(* IEC 61131-3 sources: POMIRTS_lab3/AS/Library_2/AsNxDpS, 3 files *)

(* ---- AsNxDpS.typ ---- *)
TYPE
	nxdpsAddAdrParam_t		: STRUCT			(*additional address parameter*)
		srcType				: USINT;
		srcSize				: USINT;
		destType			: USINT;
		destSize			: USINT;
		addParam			: ARRAY[0..227] OF USINT;
	END_STRUCT;

	nxdpsIm0_t				: STRUCT			(*I&M0 parameter*)
		manufactor			: ARRAY[0..9] OF USINT;
		manufactorId		: UINT;
		orderId				: ARRAY[0..19] OF USINT;
		serialNumber		: ARRAY[0..15] OF USINT;
		hwRevision			: UINT;
		swRevision			: ARRAY[0..3] OF USINT;
		revisionCounter		: UINT;
		profileId			: UINT;
		profileSpecType		: UINT;
		imVersion			: UINT;
		imSupported			: UINT;
	END_STRUCT;
END_TYPE

(* ---- AsNxDpS.fun ---- *)
{REDUND_CONTEXT} {REDUND_UNREPLICABLE} FUNCTION_BLOCK nxdpsSubscribe			(*subscribe slave*)
	VAR_INPUT
		enable			: BOOL;			(*enables execution*)
		pDevice			: UDINT;		(*interface name given as a pointer, e.g., "SL<x>.SS<y>.IF<z>"*)
	END_VAR
	VAR
        _state			: UINT;			(*internal variable*)
		_result			: UINT;			(*internal variable*)
        _srcId			: UDINT;		(*internal variable*)
	END_VAR
	VAR_OUTPUT
		status			: UINT;			(*execution status: ERR_OK, ERR_FUB_ENABLE_FALSE, ERR_FUB_BUSY, 0xXXXX = see help*)
		dpStatus		: UDINT;		(*profibus DP stack status*)
	END_VAR
END_FUNCTION_BLOCK

{REDUND_CONTEXT} {REDUND_UNREPLICABLE} FUNCTION_BLOCK nxdpsUnsubscribe			(*unsubscribe slave*)
	VAR_INPUT
		enable			: BOOL;			(*enables execution*)
		pDevice			: UDINT;		(*interface name given as a pointer, e.g., "SL<x>.SS<y>.IF<z>"*)
	END_VAR
	VAR
        _state			: UINT;			(*internal variable*)
		_result			: UINT;			(*internal variable*)
        _srcId			: UDINT;		(*internal variable*)
	END_VAR
	VAR_OUTPUT
		status			: UINT;			(*execution status: ERR_OK, ERR_FUB_ENABLE_FALSE, ERR_FUB_BUSY, 0xXXXX = see help*)
		dpStatus		: UDINT;		(*profibus DP stack status*)
	END_VAR
END_FUNCTION_BLOCK

{REDUND_CONTEXT} {REDUND_UNREPLICABLE} FUNCTION_BLOCK nxdpsAlarmNotification	(*alarm notification*)
	VAR_INPUT
		enable			: BOOL;			(*enables execution*)
		pDevice			: UDINT;		(*interface name given as a pointer, e.g., "SL<x>.SS<y>.IF<z>"*)
		slotNumber		: USINT;		(*slot number*)
		seqNumber		: USINT;		(*sequence number*)
		alarmType		: USINT;		(*alarm type*)
		alarmSpecifier	: USINT;		(*alarm specifier*)
		addAck			: BOOL;			(*additional acknowledgement flag*)
		alarmDataLen	: USINT;		(*alarm data length*)
		pAlarmData		: UDINT;		(*alarm data given as a pointer*)
	END_VAR
	VAR
        _state			: UINT;			(*internal variable*)
		_result			: UINT;			(*internal variable*)
        _srcId			: UDINT;		(*internal variable*)
	END_VAR
	VAR_OUTPUT
		status			: UINT;			(*execution status: ERR_OK, ERR_FUB_ENABLE_FALSE, ERR_FUB_BUSY, 0xXXXX = see help*)
		dpStatus		: UDINT;		(*profibus DP stack status*)
	END_VAR
END_FUNCTION_BLOCK

{REDUND_CONTEXT} {REDUND_UNREPLICABLE} FUNCTION_BLOCK nxdpsAlarmAckReceive		(*receive alarm acknowledgement*)
	VAR_INPUT
		enable			: BOOL;			(*enables execution*)
		pDevice			: UDINT;		(*interface name given as a pointer, e.g., "SL<x>.SS<y>.IF<z>"*)
	END_VAR
	VAR
        _state			: UINT;			(*internal variable*)
		_result			: UINT;			(*internal variable*)
        _srcId			: UDINT;		(*internal variable*)
	END_VAR
	VAR_OUTPUT
		status			: UINT;			(*execution status: ERR_OK, ERR_FUB_ENABLE_FALSE, ERR_FUB_BUSY, 0xXXXX = see help*)
		dpStatus		: UDINT;		(*profibus DP stack status*)
		slotNumber		: USINT;		(*slot number*)
		seqNumber		: USINT;		(*sequence number*)
		alarmType		: USINT;		(*alarm type*)
	END_VAR
END_FUNCTION_BLOCK

{REDUND_CONTEXT} {REDUND_UNREPLICABLE} FUNCTION_BLOCK nxdpsV1C1WriteInd		(*V1 class 1 write indication*)
	VAR_INPUT
		enable			: BOOL;			(*enables execution*)
		pDevice			: UDINT;		(*interface name given as a pointer, e.g., "SL<x>.SS<y>.IF<z>"*)
		maxDataLen		: UDINT;		(*max data length*)
		pData			: UDINT;		(*data buffer given as a pointer*)
	END_VAR
	VAR
        _state			: UINT;			(*internal variable*)
		_result			: UINT;			(*internal variable*)
        _srcId			: UDINT;		(*internal variable*)
	END_VAR
	VAR_OUTPUT
		status			: UINT;			(*execution status: ERR_OK, ERR_FUB_ENABLE_FALSE, ERR_FUB_BUSY, 0xXXXX = see help*)
		dpStatus		: UDINT;		(*profibus DP stack status*)
		slotNumber		: USINT;		(*slot number*)
		index			: USINT;		(*index*)
		dataLen			: USINT;		(*data length*)
		source			: UDINT;		(*source*)
		sourceId		: UDINT;		(*source id*)
	END_VAR
END_FUNCTION_BLOCK

{REDUND_CONTEXT} {REDUND_UNREPLICABLE} FUNCTION_BLOCK nxdpsV1C1WriteAck		(*V1 class 1 write acknowledgement*)
	VAR_INPUT
		enable			: BOOL;			(*enables execution*)
		pDevice			: UDINT;		(*interface name given as a pointer, e.g., "SL<x>.SS<y>.IF<z>"*)
		ackType			: BOOL;			(*type of acknowledgement*)
		slotNumber		: USINT;		(*slot number*)
		index			: USINT;		(*index*)
		dataLen			: USINT;		(*data length*)
		errorDecode		: USINT;		(*error decode*)
		errorCode1		: USINT;		(*error code 1*)
		errorCode2		: USINT;		(*error code 2*)
		source			: UDINT;		(*source*)
		sourceId		: UDINT;		(*source id*)
	END_VAR
	VAR
        _state			: UINT;			(*internal variable*)
		_result			: UINT;			(*internal variable*)
        _srcId			: UDINT;		(*internal variable*)
	END_VAR
	VAR_OUTPUT
		status			: UINT;			(*execution status: ERR_OK, ERR_FUB_ENABLE_FALSE, ERR_FUB_BUSY, 0xXXXX = see help*)
		dpStatus		: UDINT;		(*profibus DP stack status*)
	END_VAR
END_FUNCTION_BLOCK

{REDUND_CONTEXT} {REDUND_UNREPLICABLE} FUNCTION_BLOCK nxdpsV1C1ReadInd			(*V1 class 1 read indication*)
	VAR_INPUT
		enable			: BOOL;			(*enables execution*)
		pDevice			: UDINT;		(*interface name given as a pointer, e.g., "SL<x>.SS<y>.IF<z>"*)
	END_VAR
	VAR
        _state			: UINT;			(*internal variable*)
		_result			: UINT;			(*internal variable*)
        _srcId			: UDINT;		(*internal variable*)
	END_VAR
	VAR_OUTPUT
		status			: UINT;			(*execution status: ERR_OK, ERR_FUB_ENABLE_FALSE, ERR_FUB_BUSY, 0xXXXX = see help*)
		dpStatus		: UDINT;		(*profibus DP stack status*)
		slotNumber		: USINT;		(*slot number*)
		index			: USINT;		(*index*)
		dataLen			: USINT;		(*data length*)
		source			: UDINT;		(*source*)
		sourceId		: UDINT;		(*source id*)
	END_VAR
END_FUNCTION_BLOCK

{REDUND_CONTEXT} {REDUND_UNREPLICABLE} FUNCTION_BLOCK nxdpsV1C1ReadAck			(*V1 class 1 read acknowledgement*)
	VAR_INPUT
		enable			: BOOL;			(*enables execution*)
		pDevice			: UDINT;		(*interface name given as a pointer, e.g., "SL<x>.SS<y>.IF<z>"*)
		ackType			: BOOL;			(*type of acknowledgement*)
		slotNumber		: USINT;		(*slot number*)
		index			: USINT;		(*index*)
		dataLen			: USINT;		(*data length*)
		errorDecode		: USINT;		(*error decode*)
		errorCode1		: USINT;		(*error code 1*)
		errorCode2		: USINT;		(*error code 2*)
		source			: UDINT;		(*source*)
		sourceId		: UDINT;		(*source id*)
		pData			: UDINT;		(*data buffer given as pointer*)
	END_VAR
	VAR
        _state			: UINT;			(*internal variable*)
		_result			: UINT;			(*internal variable*)
        _srcId			: UDINT;		(*internal variable*)
	END_VAR
	VAR_OUTPUT
		status			: UINT;			(*execution status: ERR_OK, ERR_FUB_ENABLE_FALSE, ERR_FUB_BUSY, 0xXXXX = see help*)
		dpStatus		: UDINT;		(*profibus DP stack status*)
	END_VAR
END_FUNCTION_BLOCK

{REDUND_CONTEXT} {REDUND_UNREPLICABLE} FUNCTION_BLOCK nxdpsSetDiag				(*set diagnostic*)
	VAR_INPUT
		enable			: BOOL;			(*enables execution*)
		pDevice			: UDINT;		(*interface name given as a pointer, e.g., "SL<x>.SS<y>.IF<z>"*)
		extDiag			: BOOL;			(*extended diagnostic*)
		extDiagOverflow	: BOOL;			(*extended diagnostic overflow*)
		pDiagData		: UDINT;		(*diagnostic data given as a pointer*)
		diagDataLen		: UDINT;		(*diagnostic data length*)
	END_VAR
	VAR
        _state			: UINT;			(*internal variable*)
		_result			: UINT;			(*internal variable*)
        _srcId			: UDINT;		(*internal variable*)
	END_VAR
	VAR_OUTPUT
		status			: UINT;			(*execution status: ERR_OK, ERR_FUB_ENABLE_FALSE, ERR_FUB_BUSY, 0xXXXX = see help*)
		dpStatus		: UDINT;		(*profibus DP stack status*)
	END_VAR
END_FUNCTION_BLOCK

{REDUND_CONTEXT} {REDUND_UNREPLICABLE} FUNCTION_BLOCK nxdpsSetIm0				(*change I&M0 parameter settings*)
	VAR_INPUT
		enable				: BOOL;			(*enables execution*)
		pDevice				: UDINT;		(*interface name given as a pointer, e.g., "SL<x>.SS<y>.IF<z>"*)
		im0Param			: nxdpsIm0_t;	(*I&M0 parameter*)
		profSpecSupp		: BOOL;
		manuSpecSupp		: BOOL;
		slotsNotZeroSupp	: BOOL;
	END_VAR
	VAR
        _state			: UINT;			(*internal variable*)
		_result			: UINT;			(*internal variable*)
        _srcId			: UDINT;		(*internal variable*)
	END_VAR
	VAR_OUTPUT
		status			: UINT;			(*execution status: ERR_OK, ERR_FUB_ENABLE_FALSE, ERR_FUB_BUSY, 0xXXXX = see help*)
		dpStatus		: UDINT;		(*profibus DP stack status*)
	END_VAR
END_FUNCTION_BLOCK

{REDUND_CONTEXT} {REDUND_UNREPLICABLE} FUNCTION_BLOCK nxdpsSetAdr				(*set address*)
	VAR_INPUT
		enable			: BOOL;			(*enables execution*)
		pDevice			: UDINT;		(*interface name given as a pointer, e.g., "SL<x>.SS<y>.IF<z>"*)
		address			: UDINT;		(*new slave address*)
	END_VAR
	VAR
        _state			: UINT;			(*internal variable*)
		_result			: UINT;			(*internal variable*)
        _srcId			: UDINT;		(*internal variable*)
	END_VAR
	VAR_OUTPUT
		status			: UINT;			(*execution status: ERR_OK, ERR_FUB_ENABLE_FALSE, ERR_FUB_BUSY, 0xXXXX = see help*)
		dpStatus		: UDINT;		(*profibus DP stack status*)
	END_VAR
END_FUNCTION_BLOCK

{REDUND_CONTEXT} {REDUND_UNREPLICABLE} FUNCTION_BLOCK nxdpsStartBusComm		(*start bus communication*)
	VAR_INPUT
		enable			: BOOL;			(*enables execution*)
		pDevice			: UDINT;		(*interface name given as a pointer, e.g., "SL<x>.SS<y>.IF<z>"*)
	END_VAR
	VAR
        _state			: UINT;			(*internal variable*)
		_result			: UINT;			(*internal variable*)
        _srcId			: UDINT;		(*internal variable*)
	END_VAR
	VAR_OUTPUT
		status			: UINT;			(*execution status: ERR_OK, ERR_FUB_ENABLE_FALSE, ERR_FUB_BUSY, 0xXXXX = see help*)
		dpStatus		: UDINT;		(*profibus DP stack status*)
	END_VAR
END_FUNCTION_BLOCK

{REDUND_CONTEXT} {REDUND_UNREPLICABLE} FUNCTION_BLOCK nxdpsV1C2InitiateInd		(*V1 class2 initiate connection indication*)
	VAR_INPUT
		enable			: BOOL;			(*enables execution*)
		pDevice			: UDINT;		(*interface name given as a pointer, e.g., "SL<x>.SS<y>.IF<z>"*)
		pAddAdrParam	: UDINT;		(*additional address parameter table given as pointer*)
	END_VAR
	VAR
        _state			: UINT;			(*internal variable*)
		_result			: UINT;			(*internal variable*)
        _srcId			: UDINT;		(*internal variable*)
	END_VAR
	VAR_OUTPUT
		status			: UINT;			(*execution status: ERR_OK, ERR_FUB_ENABLE_FALSE, ERR_FUB_BUSY, 0xXXXX = see help*)
		dpStatus		: UDINT;		(*profibus DP stack status*)
		connectionRef	: UDINT;		(*connection reference*)
		featuresSup		: UINT;			(*requested featrures of the DP master class 2 connection*)
		profileFeatSup	: UINT;			(*requested profile featrures of the DP master class 2 connection*)
		profileIdent	: UINT;			(*profile ident number*)
		source			: UDINT;		(*source*)
		sourceId		: UDINT;		(*source id*)
	END_VAR
END_FUNCTION_BLOCK

{REDUND_CONTEXT} {REDUND_UNREPLICABLE} FUNCTION_BLOCK nxdpsV1C2InitiateRes		(*V1 class 2 initiate connection response*)
	VAR_INPUT
		enable			: BOOL;			(*enables execution*)
		pDevice			: UDINT;		(*interface name given as a pointer, e.g., "SL<x>.SS<y>.IF<z>"*)
		ackType			: BOOL;			(*type of acknowledgement*)
		connectionRef	: UDINT;		(*connection reference*)
		dataUnitSizeMax	: USINT;		(*maximum size of data unit to transfer*)
		featuresSup		: UINT;			(*requested featrures of the DP master class 2 connection*)
		profileFeatSup	: UINT;			(*requested profile featrures of the DP master class 2 connection*)
		profileIdent	: UINT;			(*profile ident number*)
		pAddAdrParam	: UDINT;		(*additional address parameter table given as pointer*)
		errorDecode		: USINT;		(*error decode*)
		errorCode1		: USINT;		(*error code 1*)
		errorCode2		: USINT;		(*error code 2*)
		source			: UDINT;		(*source*)
		sourceId		: UDINT;		(*source id*)
	END_VAR
	VAR
        _state			: UINT;			(*internal variable*)
		_result			: UINT;			(*internal variable*)
        _srcId			: UDINT;		(*internal variable*)
	END_VAR
	VAR_OUTPUT
		status			: UINT;			(*execution status: ERR_OK, ERR_FUB_ENABLE_FALSE, ERR_FUB_BUSY, 0xXXXX = see help*)
		dpStatus		: UDINT;		(*profibus DP stack status*)
	END_VAR
END_FUNCTION_BLOCK

{REDUND_CONTEXT} {REDUND_UNREPLICABLE} FUNCTION_BLOCK nxdpsV1C2ReadInd			(*V1 class 2 read indication*)
	VAR_INPUT
		enable			: BOOL;			(*enables execution*)
		pDevice			: UDINT;		(*interface name given as a pointer, e.g., "SL<x>.SS<y>.IF<z>"*)
	END_VAR
	VAR
        _state			: UINT;			(*internal variable*)
		_result			: UINT;			(*internal variable*)
        _srcId			: UDINT;		(*internal variable*)
	END_VAR
	VAR_OUTPUT
		status			: UINT;			(*execution status: ERR_OK, ERR_FUB_ENABLE_FALSE, ERR_FUB_BUSY, 0xXXXX = see help*)
		dpStatus		: UDINT;		(*profibus DP stack status*)
		connectionRef	: UDINT;		(*connection reference*)
		slotNumber		: USINT;		(*slot number*)
		index			: USINT;		(*index*)
		dataLen			: USINT;		(*data length*)
		source			: UDINT;		(*source*)
		sourceId		: UDINT;		(*source id*)
	END_VAR
END_FUNCTION_BLOCK

{REDUND_CONTEXT} {REDUND_UNREPLICABLE} FUNCTION_BLOCK nxdpsV1C2ReadRes			(*V1 class 2 read response*)
	VAR_INPUT
		enable			: BOOL;			(*enables execution*)
		pDevice			: UDINT;		(*interface name given as a pointer, e.g., "SL<x>.SS<y>.IF<z>"*)
		ackType			: BOOL;			(*type of acknowledgement*)
		connectionRef	: UDINT;		(*connection reference*)
		slotNumber		: USINT;		(*slot number*)
		index			: USINT;		(*index*)
		dataLen			: USINT;		(*data length*)
		errorDecode		: USINT;		(*error decode*)
		errorCode1		: USINT;		(*error code 1*)
		errorCode2		: USINT;		(*error code 2*)
		source			: UDINT;		(*source*)
		sourceId		: UDINT;		(*source id*)
		pData			: UDINT;		(*data buffer given as pointer*)
	END_VAR
	VAR
        _state			: UINT;			(*internal variable*)
		_result			: UINT;			(*internal variable*)
        _srcId			: UDINT;		(*internal variable*)
	END_VAR
	VAR_OUTPUT
		status			: UINT;			(*execution status: ERR_OK, ERR_FUB_ENABLE_FALSE, ERR_FUB_BUSY, 0xXXXX = see help*)
		dpStatus		: UDINT;		(*profibus DP stack status*)
	END_VAR
END_FUNCTION_BLOCK

{REDUND_CONTEXT} {REDUND_UNREPLICABLE} FUNCTION_BLOCK nxdpsV1C2WriteInd		(*V1 class 2 write indication*)
	VAR_INPUT
		enable			: BOOL;			(*enables execution*)
		pDevice			: UDINT;		(*interface name given as a pointer, e.g., "SL<x>.SS<y>.IF<z>"*)
		maxDataLen		: UDINT;		(*max data length*)
		pData			: UDINT;		(*data buffer given as a pointer*)
	END_VAR
	VAR
        _state			: UINT;			(*internal variable*)
		_result			: UINT;			(*internal variable*)
        _srcId			: UDINT;		(*internal variable*)
	END_VAR
	VAR_OUTPUT
		status			: UINT;			(*execution status: ERR_OK, ERR_FUB_ENABLE_FALSE, ERR_FUB_BUSY, 0xXXXX = see help*)
		dpStatus		: UDINT;		(*profibus DP stack status*)
		connectionRef	: UDINT;		(*connection reference*)
		slotNumber		: USINT;		(*slot number*)
		index			: USINT;		(*index*)
		dataLen			: USINT;		(*data length*)
		source			: UDINT;		(*source*)
		sourceId		: UDINT;		(*source id*)
	END_VAR
END_FUNCTION_BLOCK

{REDUND_CONTEXT} {REDUND_UNREPLICABLE} FUNCTION_BLOCK nxdpsV1C2WriteRes		(*V1 class 2 write response*)
	VAR_INPUT
		enable			: BOOL;			(*enables execution*)
		pDevice			: UDINT;		(*interface name given as a pointer, e.g., "SL<x>.SS<y>.IF<z>"*)
		ackType			: BOOL;			(*type of acknowledgement*)
		connectionRef	: UDINT;		(*connection reference*)
		slotNumber		: USINT;		(*slot number*)
		index			: USINT;		(*index*)
		dataLen			: USINT;		(*data length*)
		errorDecode		: USINT;		(*error decode*)
		errorCode1		: USINT;		(*error code 1*)
		errorCode2		: USINT;		(*error code 2*)
		source			: UDINT;		(*source*)
		sourceId		: UDINT;		(*source id*)
	END_VAR
	VAR
        _state			: UINT;			(*internal variable*)
		_result			: UINT;			(*internal variable*)
        _srcId			: UDINT;		(*internal variable*)
	END_VAR
	VAR_OUTPUT
		status			: UINT;			(*execution status: ERR_OK, ERR_FUB_ENABLE_FALSE, ERR_FUB_BUSY, 0xXXXX = see help*)
		dpStatus		: UDINT;		(*profibus DP stack status*)
	END_VAR
END_FUNCTION_BLOCK

{REDUND_CONTEXT} {REDUND_UNREPLICABLE} FUNCTION_BLOCK nxdpsV1C2DataInd			(*V1 class 2 data transport indication*)
	VAR_INPUT
		enable			: BOOL;			(*enables execution*)
		pDevice			: UDINT;		(*interface name given as a pointer, e.g., "SL<x>.SS<y>.IF<z>"*)
		maxDataLen		: UDINT;		(*max data length*)
		pData			: UDINT;		(*data buffer given as a pointer*)
	END_VAR
	VAR
        _state			: UINT;			(*internal variable*)
		_result			: UINT;			(*internal variable*)
        _srcId			: UDINT;		(*internal variable*)
	END_VAR
	VAR_OUTPUT
		status			: UINT;			(*execution status: ERR_OK, ERR_FUB_ENABLE_FALSE, ERR_FUB_BUSY, 0xXXXX = see help*)
		dpStatus		: UDINT;		(*profibus DP stack status*)
		connectionRef	: UDINT;		(*connection reference*)
		slotNumber		: USINT;		(*slot number*)
		index			: USINT;		(*index*)
		dataLen			: USINT;		(*data length*)
		source			: UDINT;		(*source*)
		sourceId		: UDINT;		(*source id*)
	END_VAR
END_FUNCTION_BLOCK

{REDUND_CONTEXT} {REDUND_UNREPLICABLE} FUNCTION_BLOCK nxdpsV1C2DataRes			(*V1 class 2 data transport response*)
	VAR_INPUT
		enable			: BOOL;			(*enables execution*)
		pDevice			: UDINT;		(*interface name given as a pointer, e.g., "SL<x>.SS<y>.IF<z>"*)
		ackType			: BOOL;			(*type of acknowledgement*)
		connectionRef	: UDINT;		(*connection reference*)
		slotNumber		: USINT;		(*slot number*)
		index			: USINT;		(*index*)
		dataLen			: USINT;		(*data length*)
		errorDecode		: USINT;		(*error decode*)
		errorCode1		: USINT;		(*error code 1*)
		errorCode2		: USINT;		(*error code 2*)
		source			: UDINT;		(*source*)
		sourceId		: UDINT;		(*source id*)
		pData			: UDINT;		(*data buffer given as pointer*)
	END_VAR
	VAR
        _state			: UINT;			(*internal variable*)
		_result			: UINT;			(*internal variable*)
        _srcId			: UDINT;		(*internal variable*)
	END_VAR
	VAR_OUTPUT
		status			: UINT;			(*execution status: ERR_OK, ERR_FUB_ENABLE_FALSE, ERR_FUB_BUSY, 0xXXXX = see help*)
		dpStatus		: UDINT;		(*profibus DP stack status*)
	END_VAR
END_FUNCTION_BLOCK

{REDUND_CONTEXT} {REDUND_UNREPLICABLE} FUNCTION_BLOCK nxdpsV1C2AbortInd		(*V1 class 2 abort indication*)
	VAR_INPUT
		enable			: BOOL;			(*enables execution*)
		pDevice			: UDINT;		(*interface name given as a pointer, e.g., "SL<x>.SS<y>.IF<z>"*)
	END_VAR
	VAR
        _state			: UINT;			(*internal variable*)
		_result			: UINT;			(*internal variable*)
        _srcId			: UDINT;		(*internal variable*)
	END_VAR
	VAR_OUTPUT
		status			: UINT;			(*execution status: ERR_OK, ERR_FUB_ENABLE_FALSE, ERR_FUB_BUSY, 0xXXXX = see help*)
		dpStatus		: UDINT;		(*profibus DP stack status*)
		connectionRef	: UDINT;		(*connection reference*)
		local			: UDINT;		(*local*)
		subnet			: UDINT;		(*subnet*)
		instance		: UDINT;		(*instance*)
		reasonCode		: UDINT;		(*reason code*)
		source			: UDINT;		(*source*)
		sourceId		: UDINT;		(*source id*)
	END_VAR
END_FUNCTION_BLOCK

{REDUND_CONTEXT} {REDUND_UNREPLICABLE} FUNCTION_BLOCK nxdpsV1C2AbortRes		(*V1 class 2 abort response*)
	VAR_INPUT
		enable			: BOOL;			(*enables execution*)
		pDevice			: UDINT;		(*interface name given as a pointer, e.g., "SL<x>.SS<y>.IF<z>"*)
		connectionRef	: UDINT;		(*connection reference*)
		source			: UDINT;		(*source*)
		sourceId		: UDINT;		(*source id*)
	END_VAR
	VAR
        _state			: UINT;			(*internal variable*)
		_result			: UINT;			(*internal variable*)
        _srcId			: UDINT;		(*internal variable*)
	END_VAR
	VAR_OUTPUT
		status			: UINT;			(*execution status: ERR_OK, ERR_FUB_ENABLE_FALSE, ERR_FUB_BUSY, 0xXXXX = see help*)
		dpStatus		: UDINT;		(*profibus DP stack status*)
	END_VAR
END_FUNCTION_BLOCK

(* ---- AsNxDpS.var ---- *)
VAR CONSTANT
	nxdpsERR_INVALID_DEVICE					: UINT	:= 34800;		(*error invalid device*)
	nxdpsERR_SEND_MESSAGE					: UINT	:= 34801;		(*error send message*)
	nxdpsERR_TIMEOUT						: UINT	:= 34802;		(*error timeout*)
	nxdpsERR_PROFIBUSDP_STACK				: UINT	:= 34803;		(*error receive message*)
	nxdpsERR_PARAMETER						: UINT	:= 34804;		(*error invalid parameter*)
	nxdpsERR_MEMORY							: UINT	:= 34805;		(*error less memory*)
	nxdpsERR_SUBSCRIBE_LISTENER				: UINT	:= 34806;		(*error subscribe listener*)
	nxdpsERR_NO_MORE_ENTRIES				: UINT	:= 34807;		(*error no more entries available*)

	nxdpsALARM_DIAGNOSTIC					: USINT	:= 1;			(*diagnostic alarm*)
	nxdpsALARM_PROCESS						: USINT	:= 2;			(*process alarm*)
	nxdpsALARM_PULL							: USINT	:= 3;			(*pull alarm*)
	nxdpsALARM_PLUG							: USINT	:= 4;			(*plug alarm*)
	nxdpsALARM_STATUS						: USINT	:= 5;			(*status alarm*)
	nxdpsALARM_UPDATE						: USINT	:= 6;			(*update alarm*)

	nxdpsALARM_SPEC_NO_DIFF					: USINT	:= 0;			(*no further differentiation*)
	nxdpsALARM_SPEC_ERR_APP_SLOT_DIS		: USINT	:= 1;			(*error appears and slot disturbed*)
	nxdpsALARM_SPEC_ERR_DIS_SLOT_OK			: USINT	:= 2;			(*error disappears and slot is ok*)
	nxdpsALARM_SPEC_ERR_DIS_SLOT_DIS		: USINT	:= 3;			(*error disappears and slot is still disturbed*)

	nxdpsNEGATIVE_ACK						: BOOL	:= 0;			(*negative acknowledgment*)
	nxdpsPOSITIVE_ACK						: BOOL	:= 1;			(*positive acknowledgment*)

	nxdpsMAX_DIAG_DATA_SIZE					: UDINT	:= 238;			(*max diagnostic data size*)
END_VAR
